// LS Electric XG5000 project: 0123 양솔 운전 전전후후
// PLC LSPLC

PROGRAM NewProgram (task: 스캔 프로그램)

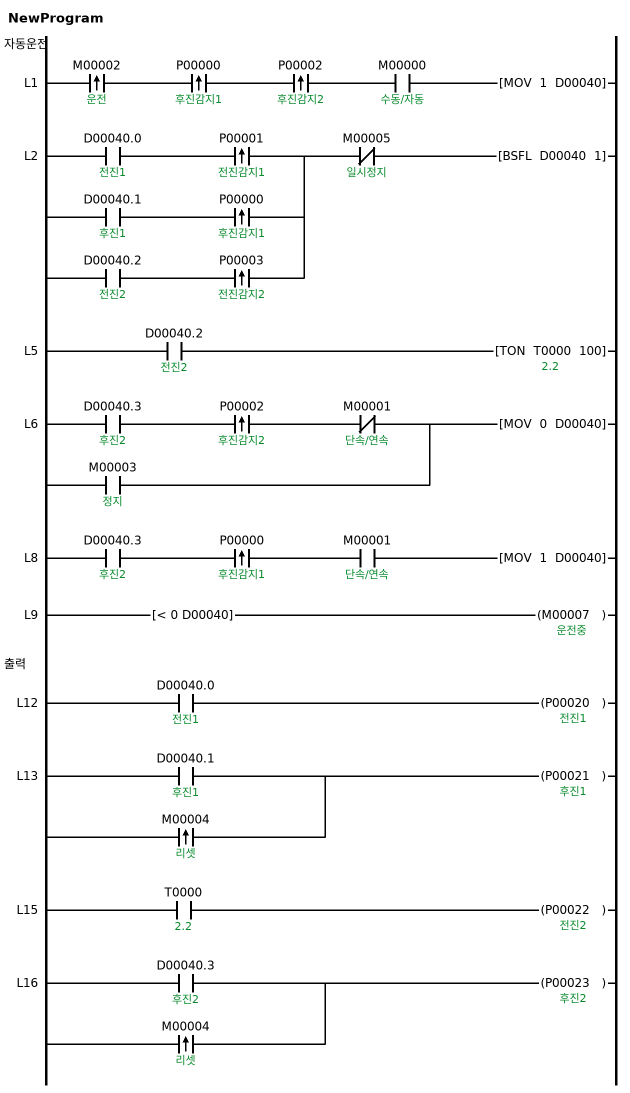
자동운전:
; L1
LOADP     M00002	// 운전
ANDP      P00000	// 후진감지1
ANDP      P00002	// 후진감지2
AND       M00000	// 수동/자동
MOV       1 D00040
; L2
LOAD      D00040.0	// 전진1
ANDP      P00001	// 전진감지1
LOAD      D00040.1	// 후진1
ANDP      P00000	// 후진감지1
OR LOAD
LOAD      D00040.2	// 전진2
ANDP      P00003	// 전진감지2
OR LOAD
AND NOT   M00005	// 일시정지
BSFL      D00040 1
; L5
LOAD      D00040.2	// 전진2
TON       T0000 100	// 2.2
; L6
LOAD      D00040.3	// 후진2
ANDP      P00002	// 후진감지2
AND NOT   M00001	// 단속/연속
OR        M00003	// 정지
MOV       0 D00040
; L8
LOAD      D00040.3	// 후진2
ANDP      P00000	// 후진감지1
AND       M00001	// 단속/연속
MOV       1 D00040
; L9
LOAD<     0 D00040
OUT       M00007	// 운전중
출력:
; L12
LOAD      D00040.0	// 전진1
OUT       P00020	// 전진1
; L13
LOAD      D00040.1	// 후진1
ORP       M00004	// 리셋
OUT       P00021	// 후진1
; L15
LOAD      T0000	// 2.2
OUT       P00022	// 전진2
; L16
LOAD      D00040.3	// 후진2
ORP       M00004	// 리셋
OUT       P00023	// 후진2